PROGRAM MAIN
VAR
	open_directive		: 	BOOL;
	delay 				:	LINT;
	delay_timer_limit	:	LINT;
	open_pin 	AT%Q* 	: 	BOOL;
	close_pin 	AT%Q* 	:	BOOL;
	
	open_limit 	AT%I*	: 	BOOL;
	close_limit AT%I*	: 	BOOL;
END_VAR


IF NOT open_directive THEN
	IF delay < delay_timer_limit THEN
		delay := delay+ 1;
	END_IF
ELSE
	delay := 0;
END_IF

IF delay >= delay_timer_limit THEN
	close_pin := TRUE;
ELSE
	close_pin := FALSE;
END_IF

open_pin := open_directive;
(*
IF NOT open_limit THEN
	open_pin := open_directive;
ELSE
	open_PIN := FALSE;
END_IF
*)

END_PROGRAM

(* stored: Version 1.1.0.1, ProductVersion 3.1.4024.0
   POU MAIN: Id {e29008e8-7ba7-4a55-838a-88b2f90948ea}, SpecialFunc None *)
